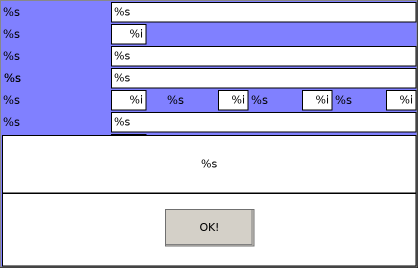
VISUALIZATION VISU_INFO_PROCESS  // 418x268
    Rectangle (0,0 418x268)
    Button (296,202 120x30), "%s", input disabled if: NOT (PRG_USER.ACTU_USER.PRODUCTION), text list: 'TextList_Process', text index: 26
        toggle EXECPROC.M_LOAD_PROCESS
    Rectangle (0,2 110x20), "%s", text list: 'TextList_Process', text index: 7
    Rectangle (111,2 305x20), "%s", text variable: EXECPROC.PRM_PROCESS
    Rectangle (0,24 110x20), "%s", text list: 'TextList_Process', text index: 8
    Rectangle (111,24 35x20), "%i", text variable: EXECPROC.STATE_STEP
    Rectangle (0,46 110x20), "%s", text list: 'TextList_Process', text index: 9
    Rectangle (111,46 305x20), "%s", text list: 'TextList_Type_Etape', text index: EXECPROC.PRM_TYPE_ETAPE
    Rectangle (0,90 110x20), "%s", invisible if: MAIN.STEP_EMPILEMENT.OP_RUN.AR, text list: 'TextList_Process', text index: 11
    Rectangle (111,90 35x20), "%i", text variable: MAIN.STEP_EMPILEMENT.STATE_LAYER, invisible if: MAIN.STEP_EMPILEMENT.OP_RUN.AR
    Rectangle (0,112 110x20), "%s", invisible if: MAIN.STEP_EMPILEMENT.OP_RUN.AR, text list: 'TextList_Process', text index: 12
    Rectangle (111,112 305x20), "%s", text variable: MAIN.STEP_EMPILEMENT.STATE_LAYER_TEXT, invisible if: MAIN.STEP_EMPILEMENT.OP_RUN.AR
    Rectangle (164,90 55x20), "%s", invisible if: MAIN.STEP_EMPILEMENT.OP_RUN.AR OR (MAIN.STEP_EMPILEMENT.PRM_NB_LOOP = 0), text list: 'TextList_Process', text index: 13
    Rectangle (248,90 55x20), "%s", invisible if: MAIN.STEP_EMPILEMENT.OP_RUN.AR OR (MAIN.STEP_EMPILEMENT.PRM_NB_LOOP = 0), text list: 'TextList_Process', text index: 14
    Rectangle (218,90 30x20), "%i", text variable: MAIN.STEP_EMPILEMENT.PRM_NB_LOOP, invisible if: MAIN.STEP_EMPILEMENT.OP_RUN.AR OR (MAIN.STEP_EMPILEMENT.PRM_NB_LOOP = 0)
    Rectangle (302,90 30x20), "%i", text variable: MAIN.STEP_EMPILEMENT.PRM_LOOP_FIRST_LAYER, invisible if: MAIN.STEP_EMPILEMENT.OP_RUN.AR OR (MAIN.STEP_EMPILEMENT.PRM_NB_LOOP = 0)
    Rectangle (332,90 55x20), "%s", invisible if: MAIN.STEP_EMPILEMENT.OP_RUN.AR OR (MAIN.STEP_EMPILEMENT.PRM_NB_LOOP = 0), text list: 'TextList_Process', text index: 15
    Rectangle (386,90 30x20), "%i", text variable: MAIN.STEP_EMPILEMENT.PRM_LOOP_LAST_LAYER, invisible if: MAIN.STEP_EMPILEMENT.OP_RUN.AR OR (MAIN.STEP_EMPILEMENT.PRM_NB_LOOP = 0)
    Rectangle (0,134 110x20), "%s", invisible if: PRG_EVAP.EVAPS1.OP_Marche.AR, text list: 'TextList_Process', text index: 16
    Rectangle (0,156 110x20), "%s", invisible if: PRG_EVAP.EVAPS1.OP_Marche.AR, text list: 'TextList_Process', text index: 17
    Rectangle (0,178 110x20), "%s", invisible if: PRG_EVAP.EVAPS1.OP_Marche.AR, text list: 'TextList_Process', text index: 18
    Rectangle (111,134 35x20), "%i", text variable: PRG_EVAP.EVAPS1.STATE_Segment, invisible if: PRG_EVAP.EVAPS1.OP_Marche.AR
    Rectangle (111,156 305x20), "%s", text variable: PRG_EVAP.EVAPS1.STATE_Temps_segment, invisible if: PRG_EVAP.EVAPS1.OP_Marche.AR
    Rectangle (111,178 305x20), "%s", text variable: PRG_EVAP.EVAPS1.TIMER_Temps_Couche.ET, invisible if: PRG_EVAP.EVAPS1.OP_Marche.AR, text index: 18
    Button (149,202 120x30), "%s", input disabled if: NOT (PRG_USER.ACTU_USER.PRODUCTION AND MAIN.STEP_EMPILEMENT.AUTOR_NEXT_LAYER), text list: 'TextList_Process', text index: 19
        toggle MAIN.STEP_EMPILEMENT.M_NEXT_LAYER
    Button (2,234 120x30), "%s", input disabled if: NOT (PRG_USER.ACTU_USER.PRODUCTION AND MACHINE.AUTOR_Inter_Prod_ihm), text list: 'TextList_Process', text index: 20
        toggle MACHINE.M_inter_Prod
    Button (149,234 120x30), "%s", input disabled if: NOT (PRG_USER.ACTU_USER.PRODUCTION AND MACHINE.AUTOR_Repris_Prod_ihm), text list: 'TextList_Process', text index: 21
        toggle MACHINE.M_Reprise_Prod
    Button (296,234 120x30), "%s", input disabled if: NOT (PRG_USER.ACTU_USER.PRODUCTION AND MACHINE.AUTOR_Stop_Prod_Ihm), text list: 'TextList_Process', text index: 22
        toggle MACHINE.M_Stop_Prod
    Button (2,202 120x30), "%s", input disabled if: NOT (PRG_USER.ACTU_USER.PRODUCTION AND EXECPROC.AUTOR_NEXT_STEP), text list: 'TextList_Process', text index: 23
        toggle EXECPROC.M_NEXT_STEP
    Rectangle (111,68 305x20), "/", invisible if: NOT MAIN.STEP_TIMER.I_ON
    Rectangle (126,69 121x18), "%s", text variable: MAIN.STEP_TIMER.TIMER.ET, invisible if: NOT MAIN.STEP_TIMER.I_ON
    Rectangle (288,69 121x18), "%s", text variable: MAIN.STEP_TIMER.TIMER.PT, invisible if: NOT MAIN.STEP_TIMER.I_ON
    Rectangle (1,68 110x20), "%s", invisible if: NOT EXECPROC.RQ_EXEC_STEP[1], text list: 'TextList_Process', text index: 12
    Rectangle (111,68 305x20), "%s", text variable: PRG_POMPAGE.PRM_Pr_Pumping_OK, invisible if: NOT EXECPROC.RQ_EXEC_STEP[1]
    Rectangle (0,179 110x20), "%s", invisible if: PRG_EVAP.EVAPS2.OP_Marche.AR, text list: 'TextList_Process', text index: 18
    Rectangle (0,135 110x20), "%s", invisible if: PRG_EVAP.EVAPS2.OP_Marche.AR, text list: 'TextList_Process', text index: 16
    Rectangle (0,157 110x20), "%s", invisible if: PRG_EVAP.EVAPS2.OP_Marche.AR, text list: 'TextList_Process', text index: 17
    Rectangle (111,135 35x20), "%i", text variable: PRG_EVAP.EVAPS2.STATE_Segment, invisible if: PRG_EVAP.EVAPS2.OP_Marche.AR
    Rectangle (111,157 305x20), "%s", text variable: PRG_EVAP.EVAPS2.STATE_Temps_segment, invisible if: PRG_EVAP.EVAPS2.OP_Marche.AR
    Rectangle (111,179 305x20), "%s", text variable: PRG_EVAP.EVAPS2.TIMER_Temps_Couche.ET, invisible if: PRG_EVAP.EVAPS2.OP_Marche.AR, text index: 18
    Rectangle (0,178 110x20), "%s", invisible if: PRG_EVAP.EVAPS3.OP_Marche.AR, text list: 'TextList_Process', text index: 18
    Rectangle (0,134 110x20), "%s", invisible if: PRG_EVAP.EVAPS3.OP_Marche.AR, text list: 'TextList_Process', text index: 16
    Rectangle (0,156 110x20), "%s", invisible if: PRG_EVAP.EVAPS3.OP_Marche.AR, text list: 'TextList_Process', text index: 17
    Rectangle (111,134 35x20), "%i", text variable: PRG_EVAP.EVAPS3.STATE_Segment, invisible if: PRG_EVAP.EVAPS3.OP_Marche.AR
    Rectangle (111,156 305x20), "%s", text variable: PRG_EVAP.EVAPS3.STATE_Temps_segment, invisible if: PRG_EVAP.EVAPS3.OP_Marche.AR
    Rectangle (111,178 305x20), "%s", text variable: PRG_EVAP.EVAPS3.TIMER_Temps_Couche.ET, invisible if: PRG_EVAP.EVAPS3.OP_Marche.AR, text index: 18
    Rectangle (2,193 414x73), invisible if: NOT MAIN.STEP_USER_ACK.STATE_EC
    Button (165,209 89x37), "OK!", invisible if: NOT MAIN.STEP_USER_ACK.STATE_EC
        tap MAIN.STEP_USER_ACK.M_GOON
    Rectangle (2,135 414x58), "%s", text variable: MAIN.STEP_USER_ACK.PRM_TEXT, invisible if: NOT MAIN.STEP_USER_ACK.STATE_EC
    Rectangle (1,68 110x20), "%s", invisible if: MAIN.STEP_EFFLUVAGE.OP_RUN.AR or true, text list: 'TextList_Process', text index: 10
END_VISUALIZATION

(* stored: Version 1.1.0.1, ProductVersion 3.1.4024.12
   Visu VISU_INFO_PROCESS: Id {8e2c49f8-7329-4f39-bb8c-eace05072c2b} *)
